// TIA Portal V15.1 export
// export: Created 2024-05-17T05:38:12.2995239Z, ExportSetting WithDefaults, DisplayName Totally Integrated Automation Portal, DisplayVersion V15.1 Update 5, DisplayName TIA Portal Openness, DisplayVersion V15.1 Update 5, DisplayName SINAMICS Startdrive Advanced, DisplayVersion V15.1, DisplayName G130, G150, S120, S150, SINAMICS MV, S210, DisplayVersion V15.1, DisplayName G110M, G120, G120C, G120D, G120P, DisplayVersion V15.1, DisplayName STEP 7 Professional, DisplayVersion V15.1 Update 5, DisplayName STEP 7 Safety, DisplayVersion V15.1, DisplayName WinCC Professional, DisplayVersion V15.1 Update 5, DisplayName SIMATIC Visualization Architect, DisplayVersion V15.1
DATA_BLOCK "_209000NCP01PNIODiagList"   // DB271
{ S7_Optimized_Access := 'TRUE' }
AUTHOR : VCC
VERSION : 0.1
// stored: AutoNumber false, DBAccessibleFromOPCUA true, IsOnlyStoredInLoadMemory false, IsRetainMemResEnabled false, IsWriteProtectedInAS false, MemoryReserve 0
   VAR
      PNIODiag_StartFillList { ExternalAccessible := 'False'; ExternalVisible := 'False'; ExternalWritable := 'False'} : Bool;   // PNIODiag - Start with fill-in the list
      PNIODiag_LastDeviceNumber { ExternalAccessible := 'False'; ExternalVisible := 'False'; ExternalWritable := 'False'} : Int;   // PNIODiag - Last Device Number
      PNIODiag_ListIPDone { ExternalAccessible := 'False'; ExternalVisible := 'False'; ExternalWritable := 'False'} : Bool;   // PNIODiag - The list with the IP adress is done
      PNIODiag_ListMACDone { ExternalAccessible := 'False'; ExternalVisible := 'False'; ExternalWritable := 'False'} : Bool;   // PNIODiag - The list with the MAC adress is done
      PNIODiag_ListNameDone { ExternalAccessible := 'False'; ExternalVisible := 'False'; ExternalWritable := 'False'} : Bool;   // PNIODiag - The list with the Profinet name is done
      PNIODiag_ListAllDone { ExternalAccessible := 'False'; ExternalVisible := 'False'; ExternalWritable := 'False'} : Bool;   // PNIODiag - All lists are done
      PNIODiag_ListBusy { ExternalAccessible := 'False'; ExternalVisible := 'False'; ExternalWritable := 'False'} : Bool;   // PNIODiag - Busy with fill in of the lists
      PNIODiag_DeviceExist { ExternalAccessible := 'False'; ExternalVisible := 'False'; ExternalWritable := 'False'} : Array[0..255] of Bool;   // PNIODiag - List with existing devices
      PNIODiag_HWIdentifier { ExternalAccessible := 'False'; ExternalVisible := 'False'; ExternalWritable := 'False'} : Array[0..255] of UInt;   // PNIODiag - List with hardware indentifier from each device
      PNIODiag_GetStationName { ExternalAccessible := 'False'; ExternalVisible := 'False'; ExternalWritable := 'False'} : Array[0..255] of String;   // PNIODiag - List with Profinet name from each device
      PNIODiag_GetStationIP { ExternalAccessible := 'False'; ExternalVisible := 'False'; ExternalWritable := 'False'} : Array[0..255] of IF_CONF_v4;   // PNIODiag - List with IP adress from each device
      PNIODiag_GetStationMAC { ExternalAccessible := 'False'; ExternalVisible := 'False'; ExternalWritable := 'False'} : Array[0..255] of IF_CONF_MAC;   // PNIODiag - List with MAC adress from each device
      PNIODiag_Global { ExternalAccessible := 'False'; ExternalVisible := 'False'; ExternalWritable := 'False'} : "H_PNIODiagS7-1500";   // PNIODIAG - HMI
      PNIODiag_ListStationName { ExternalAccessible := 'False'; ExternalVisible := 'False'; ExternalWritable := 'False'} : Array[0..255] of String[25];   // PNIODIAG - HMI list
      PNIODiag_ListIPAddress { ExternalAccessible := 'False'; ExternalVisible := 'False'; ExternalWritable := 'False'} : Array[0..255] of String[15];   // PNIODIAG - HMI list
      PNIODiag_ListMACAddress { ExternalAccessible := 'False'; ExternalVisible := 'False'; ExternalWritable := 'False'} : Array[0..255] of String[18];   // PNIODIAG - HMI list
      Edge001 { ExternalAccessible := 'False'; ExternalVisible := 'False'; ExternalWritable := 'False'} : Bool;   // Edge
      Edge002 { ExternalAccessible := 'False'; ExternalVisible := 'False'; ExternalWritable := 'False'} : Bool;   // Edge
   END_VAR
BEGIN
END_DATA_BLOCK
